TYPE ST_IngotPrevent :
STRUCT
	biSnIngotPrevent_Forward:BOOL;
	biSnIngotPrevent_Back:BOOL;
	BoCylIngotPrevent_Forward:BOOL;
	BoCylIngotPrevent_Back:BOOL;
	biSnIngotPreventBtn_Forward:BOOL;
	biSnIngotPreventBtn_Back:BOOL;
END_STRUCT
END_TYPE

(* stored: Version 1.1.0.1, ProductVersion 3.1.4024.12
   DUT ST_IngotPrevent: Id {89374f60-d1af-42d8-87d2-f9c29a3303fd} *)
